//Test suite for the FB_Axis POU
{attribute 'call_after_init'}
FUNCTION_BLOCK FB_Axis_TEST EXTENDS tcUnit.FB_TestSuite
VAR
    fbCommon: FB_tcUNIT_common;
    iTargetAxis: UINT := 1; //The <index> of the axis within GVL.astAxes[<index>] to test against.
END_VAR

//Declare methods defined in the FB_Axis_TEST POU to be included (executed) in the test suite
SetAxisControl_Enabled();
CheckAxisStatus_Moving();
SetAxisConfig_Acceleration();
CheckAxisStatus_NewPosition();
SetAxisControl_Velocity();
SetAxisInputs_bLimitFwd();

METHOD CheckAxisStatus_Moving
VAR
    Result: BOOL;
    ExpectedResult: BOOL;

    nCycle: UINT;
    nMaxCycles: UINT := 30;
END_VAR
TEST('test_GIVEN_new_axis_position_WHEN_execute_move_THEN_axis_moves');

ExpectedResult := TRUE;

fbCommon.mPrepareDefaultMove(iTargetAxis);
fbCommon.mExecute(iTargetAxis);

Result := GVL.astAxes[iTargetAxis].stStatus.bBusy;

IF nCycle > nMaxCycles OR ExpectedResult = Result THEN
    AssertEquals(Expected := ExpectedResult,
                 Actual := Result,
                 Message := 'Axis is not moving.');
    TEST_FINISHED();
ELSE
    nCycle := nCycle + 1;
END_IF
END_METHOD

METHOD CheckAxisStatus_NewPosition
VAR
    InitialValue: LREAL;
    Result: LREAL;
    ExpectedResult: LREAL;

    nCycle: UINT;
    nCycleMax: UINT := 100;
END_VAR
TEST('test_GIVEN_new_axis_position_set_WHEN_executed_THEN_axis_moves_to_new_position');

//Since the axis has state; a test might begin the position at some location set by
//a previous test. Therefore if we execute a move we should just check it's moved
//from the initial location not some initial default.

InitialValue := GVL.astAxes[iTargetAxis].stConfig.fPosition;
ExpectedResult := InitialValue + 10;
GVL.astAxes[iTargetAxis].stConfig.fPosition := ExpectedResult;

GVL.astAxes[iTargetAxis].stControl.eCommand := E_MotionFunctions.eMoveAbsolute;
GVL.astAxes[iTargetAxis].stControl.bExecute := TRUE;

Result := GVL.astAxes[iTargetAxis].stStatus.fActPosition;

IF nCycle > nCycleMax OR ExpectedResult = Result THEN
    AssertEquals(Expected := ExpectedResult,
                 Actual := Result,
                 Message := 'fPosition of the axis is different.');
    TEST_FINISHED();
ELSE
    nCycle := nCycle + 1;
END_IF
END_METHOD

METHOD SetAxisConfig_Acceleration
VAR
    InitialValue: LREAL;
    Result: LREAL;
    ExpectedResult: LREAL;
END_VAR
TEST('test_GIVEN_new_axis_acceleration_set_WHEN_executed_THEN_new_axis_acceleration_set');

//example of direct GVL axis reference for assert.

ExpectedResult := tcUNIT_gvl.fDEFAULT_TARGET_ACCELERATION;
fbCommon.mPrepareDefaultMove(iTargetAxis);

Result := GVL.astAxes[iTargetAxis].stConfig.fAcceleration;

AssertEquals(Expected := ExpectedResult,
             Actual := Result,
             Message := 'fAcceleration of the axis is different.');

TEST_FINISHED();
END_METHOD

METHOD SetAxisControl_Enabled
VAR
    Result: BOOL;
    ExpectedResult: BOOL;

    nCycle: UINT;
    nMaxCycles: UINT := 30;
END_VAR
TEST('test_GIVEN_prepare_default_move_WHEN_move_prepared_THEN_axis_enabled');

//example of test that requires multiple cycles to complete. Due to stateful behaviour of the axis structure.

ExpectedResult := TRUE;
GVL.astAxes[iTargetAxis].stControl.bEnable := ExpectedResult;

Result := GVL.astAxes[iTargetAxis].stStatus.bEnabled;

IF nCycle > nMaxCycles OR ExpectedResult = Result THEN
    AssertEquals(Expected := ExpectedResult,
                 Actual := Result,
                 Message := 'Axis is not enabled.');
    TEST_FINISHED();
ELSE
    nCycle := nCycle + 1;
END_IF
END_METHOD

METHOD SetAxisControl_Velocity
VAR
    InitialValue: LREAL;
    Result: LREAL;
    ExpectedResult: LREAL;

    fDelta: REAL := 0.01;
END_VAR
TEST('test_GIVEN_new_axis_velocity_set_WHEN_executed_THEN_new_axis_velocity_set');

//Example of using a tcUNIT assert for a specific type (in this case LREAL).

InitialValue := GVL.astAxes[iTargetAxis].stConfig.fVelocity;
ExpectedResult := InitialValue + 0.5;
GVL.astAxes[iTargetAxis].stConfig.fVelocity := ExpectedResult;

Result := GVL.astAxes[iTargetAxis].stConfig.fVelocity;

AssertEquals_LREAL(Expected := ExpectedResult,
                   Actual := Result,
                   Delta := fDelta,
                   Message := 'fVelocity of the axis is different.');
    TEST_FINISHED();
END_METHOD

METHOD SetAxisInputs_bLimitFwd
VAR
    Result: BOOL;
    ExpectedResult: BOOL;

    nCycle: UINT;
    nMaxCycles: UINT := 30;
END_VAR
TEST('test_GIVEN_prepare_default_move_WHEN_bFwEnabled_prepared_enabled_THEN_bFwEnable_enabled');

ExpectedResult := TRUE;

GVL.astAxes[iTargetAxis].stInputs.bLimitFwd := TRUE;

Result := GVL.astAxes[iTargetAxis].stStatus.bFwEnabled;

IF nCycle > nMaxCycles OR ExpectedResult = Result THEN
    AssertEquals(Expected := ExpectedResult,
                 Actual := Result,
                 Message := 'Axis bLimitFwd is not enabled.');
    TEST_FINISHED();
ELSE
    nCycle := nCycle + 1;
END_IF
END_METHOD

END_FUNCTION_BLOCK

(* stored: Version 1.1.0.1, ProductVersion 3.1.4024.5
   POU FB_Axis_TEST: Id {3bfca2b4-3b3f-48f2-9900-9d4cd3404e9e}, SpecialFunc None
   Method CheckAxisStatus_Moving: Id {f7dcf822-91ec-4555-918f-e2487353578a}
   Method CheckAxisStatus_NewPosition: Id {604b9446-af57-41db-afac-f53f5b12cc2c}
   Method SetAxisConfig_Acceleration: Id {2efd2402-6ad3-455d-a703-347847c98522}
   Method SetAxisControl_Enabled: Id {749049e6-6152-4a23-ac76-75883bd089b7}
   Method SetAxisControl_Velocity: Id {f87270b6-fb94-4214-bb13-17f22f6ab8f5}
   Method SetAxisInputs_bLimitFwd: Id {6304c3b1-9e72-403e-9ae2-a5609b1efe92} *)
